FUNCTION_BLOCK OPCUA_BOOL_VARIABLE_LISTENER
  {SET_ATTRIBUTE(OpcUa, POINT.STARTPOINT)}
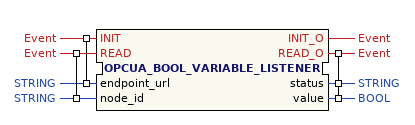
  EVENT_INPUT
    INIT WITH endpoint_url;
    READ WITH node_id; {SET_ATTRIBUTE(OpcUa, Method)}
  END_EVENT
  EVENT_OUTPUT
    INIT_O;
    READ_O WITH status, value;
  END_EVENT
  VAR_INPUT
    endpoint_url : STRING; {SET_ATTRIBUTE(OpcUa, Constant.RUN)}
    node_id : STRING; {SET_ATTRIBUTE(OpcUa, Variable.RUN)}
  END_VAR
  VAR_OUTPUT
    status : STRING; {SET_ATTRIBUTE(OpcUa, Variable.RUN)}
    value : BOOL; {SET_ATTRIBUTE(OpcUa, Variable.RUN)}
  END_VAR
END_FUNCTION_BLOCK
